TYPE T_DataType : PVOID; END_TYPE

(* stored: Version 1.1.0.1, ProductVersion 3.1.4024.12
   DUT T_DataType: Id {11f982fd-c627-41e6-852b-5da396a9cbcb} *)
